# B&R Automation Studio project server
Automation Studio 4.4.6.71 SP

## Configuration minimal

### Hardware
```
X20CP1586 : X20CP1586 v1.4.2.0
  Connector IF2:
    ActivateDevice = 1
    Mode = Manual
    InternetAddress = 10.4.22.176
    SubnetMask = 255.255.255.0
  ConfigurationID = br_server_minimal
  Simulation = 1
```

## Logical view

Binary libraries used (declarations not repeated): AsBrStr, AsIecCon, AsIOTime, runtime

### Global.typ - Global data types
```iecst
TYPE
	_expData : 	STRUCT
		bActivateExperiment : BOOL;
	END_STRUCT;
	_trajData : 	STRUCT
		dStartValue : LREAL;
		lStartTime : UDINT;
		dEndValue : LREAL;
		lEndTime : UDINT;
		dOutput : LREAL;
	END_STRUCT;
	_benchData : 	STRUCT
		lTime : UDINT;
		dValue1 : LREAL;
		fValue2 : REAL;
		iValue3 : INT;
		cValue4 : BYTE;
		dValueNan : LREAL;
		dValueInf : LREAL;
	END_STRUCT;
END_TYPE
```

### Global.var - Global variables
```iecst
VAR
	expData : _expData;
	trajData : _trajData;
	benchData : _benchData;
END_VAR
```

### Package Logical/Libraries - Global libraries

### Comm.h
```c
/**
 * @file Comm.h
 */
#ifndef COMM_H
#define COMM_H

#include "Transport/Frame.h"

#define MAX_PAYLOAD (80)

/**
 * @class Comm
 * @brief defines an interface class which lets the TcpIpServer communicate with the transport protocol
 */
class Comm {
	public:
	virtual void handleFrame(Frame frame) = 0;
};

#endif
```

### TcpIpServer.h
```c
#ifndef TCPSERVER_CLASS_H
#define TCPSERVER_CLASS_H
#include <bur/plctypes.h>
#ifdef _DEFAULT_INCLUDES
#include <AsDefault.h>
#endif
#include <AsTCP.h>
#include <AsIOTime.h>
#include "../Comm.h"
#include "../Transport/Frame.h"

/** @file TcpServer.h
 *  @class TcpIpServer
 *  @brief Implementation of a simple TCP Server
 *
 *	The server is initialised and run using the BuR AsTCP library.
 */

class TcpIpServer: public Comm{
	public:
	/** server status enum */
	enum Status
	{
		ERROR = 0xFF,
		STOP = 0,
		BUSY,
		READY
	};
	private:
	const int serverPort;		///< port to be used by the server
	unsigned long serverID;		///< server ID for function blocks

	unsigned long clientIp;		///< IP address of connected client
	unsigned long clientID;		///< client ID for function blocks

	unsigned short tcp_step;		///< step variable for the server state-machine

	Status _status;
	Status _status_sub;

	struct TcpOpen TcpOpen_0;
	struct TcpServer TcpServer_0;
	struct TcpIoctl TcpIoctl_0;
	struct TcpRecv TcpRecv_0;
	struct TcpSend TcpSend_0;
	struct TcpClose TcpClose_0;

	unsigned char outBuffer[2][255 * (MAX_PAYLOAD + 1)];
	unsigned int outBufferLen[2];
	unsigned char currentOutBuf;
	unsigned char inBuffer[255 * (MAX_PAYLOAD + 1)];
	unsigned int inBufferLen;

	Status read();
	Status write();

	Comm *transp;

	public:
	TcpIpServer(int port)
		:serverPort(port),
		status(_status)
	{};

	void deinit();
	void init();
	/** cyclic read/write method */
	void sync();

	void closeSockets();
	/** readonly pointer to server status */
	const Status &status;
	/** Method to queue communication frame */
	void handleFrame(Frame frame);
	/** Method to register the transport protocol instance */
	void registerListener(Comm *transp);
};
#endif //TCPSERVER_CLASS_H
```

### Program Logical/Libraries/Transport

#### Frame.h
```c
/** @file Frame.h
 *
 */
#ifndef FRAME_H
#define FRAME_H

#include <bur/plctypes.h>
#ifdef _DEFAULT_INCLUDES
#include <AsDefault.h>
#endif
#include <stdint.h>
#include <assert.h>
#include <stdio.h>
#include <string.h>

#include "../Comm.h"

/** frame length */
#define MAX_PAYLOAD (80)

/**
 * Class, that implements a byte wise frame that is interchanged by connection. The frame has an id and a payload
 * for the specific data. The data is stored as an byte array. It implements all functions to store and unpack
 * the data to and from byte wise array. The id represents the identification of the frame.
 */
class Frame {

public:
	struct _data {
		unsigned char id;
		unsigned char payload[80];
	} data;

	Frame(unsigned char id) {
		data.id = id;
		cCursor = 0;
	}

	Frame() {
		cCursor = 0;
	}

    /** pack value into Frame
     *
     * use `pack<typename>(value)` to be explicit
     **/
	template<typename T>
	void pack(T value) {
		const unsigned int sz = sizeof(T);
		assert(cCursor + sz < MAX_PAYLOAD);
		memcpy(&data.payload[cCursor], &value, sz);
		cCursor += sz;
	}

	/** unpack into value from Frame
     *
     * use `unPack<typename>(location)` to be explicit
     */
	template<typename T>
	void unPack(T &value) {
		const unsigned int sz = sizeof(T);
		assert(cCursor + sz < MAX_PAYLOAD);
		memcpy(&value, &data.payload[cCursor], sz);
		cCursor += sz;
	}

private:
	unsigned char cCursor;

	union {
		double dVar;
		struct {
			float fVar2;
			float fVar1;
		};
		unsigned char cVar[8];
	} uPack;

};

#endif //SERVER_FRAME_H
```

#### Transport.cpp
```cpp
#define _BUR_USE_DECLARATION_IN_IEC
#ifdef _DEFAULT_INCLUDES
#include "AsDefault.h"
#endif
#include "Transport.h"

/**
 * @brief Method that defines and sends all testbench frames
 */
void Transport::sendData() {
	Frame benchFrame(10);
	benchFrame.pack(benchData.lTime);
	benchFrame.pack(benchData.dValue1);
	benchFrame.pack(benchData.fValue2);
	benchFrame.pack(benchData.iValue3);
	benchFrame.pack(benchData.cValue4);
	benchFrame.pack(benchData.dValueNan);
	benchFrame.pack(benchData.dValueInf);
	tcp->handleFrame(benchFrame);

	Frame trajFrame(11);
	trajFrame.pack(benchData.lTime);
	trajFrame.pack(trajData.dOutput);
	tcp->handleFrame(trajFrame);
}

/*
 * @brief handles all frames arriving at the testbench
 */
void Transport::handleFrame(Frame frame)
{
	switch (frame.data.id) {
		case 1:
			unpackExp(frame);
			break;
		case 12:
			unpackBenchData(frame);
			break;
		case 13:
			unpackTrajRampData(frame);
			break;
		default:;
	}
}

/**
 * @brief unpacks experiment activation status and resets experiment time
 */
void Transport::unpackExp(Frame frame) {
	frame.unPack(expData.bActivateExperiment);
	benchData.lTime = 0;
}

void Transport::unpackBenchData(Frame frame) {
	frame.unPack(benchData.dValue1);
	frame.unPack(benchData.fValue2);
	frame.unPack(benchData.iValue3);
	frame.unPack(benchData.cValue4);
}

void Transport::unpackTrajRampData(Frame frame) {
	frame.unPack(trajData.dStartValue);
	frame.unPack(trajData.lStartTime);
	frame.unPack(trajData.dEndValue);
	frame.unPack(trajData.lEndTime);
}

/**
 * @brief registers Server for handling outgoing frames
 */
void Transport::registerServer(Comm *serv)
{
	this->tcp = serv;
}
```

### Program Logical/ControlLoop (ANSIC)

#### Main.cpp - Init, cyclic, exit code
```cpp
#include <bur/plc.h>
#include <bur/plctypes.h>
#include <math.h>

#ifdef _DEFAULT_INCLUDES
	#include <AsDefault.h>
#endif

#include "../Libraries/Transport/Transport.h"

// amount of memory to be allocated for heap storage must be specified for every ANSI C++ program with the bur_heap_size variable
unsigned long bur_heap_size = 0xFFFF;
const unsigned long lDt = 1000;          ///< Sampling step [ms]

/**
 * @brief Method that calculates a trajectory value and writes the return value in _trajData->dOutput
 * @param _benchData pointer to test rig data struct
 * @param _trajData pointer to trajectory struct
 */
void fTrajectory() {
	if (benchData.lTime < trajData.lStartTime) {
		trajData.dOutput = trajData.dStartValue;
	} else {
		if (benchData.lTime < trajData.lEndTime) {
			double dM = (trajData.dEndValue - trajData.dStartValue) / (trajData.lEndTime - trajData.lStartTime);
			double dN = trajData.dEndValue - dM * trajData.lEndTime;
			trajData.dOutput = dM * benchData.lTime + dN;
		} else {
			trajData.dOutput = trajData.dEndValue;
		}
	}
}

void _INIT ProgramInit(void) {
	benchData.lTime = 0;
	benchData.dValue1 = 0;
	benchData.fValue2 = 0;
	benchData.iValue3 = 0;
	benchData.cValue4 = 0;
	benchData.dValueNan = nan("");
	benchData.dValueInf =  infinity();

	trajData.dStartValue = 0;
	trajData.lStartTime = 0;
	trajData.dEndValue = 0;
	trajData.lEndTime = 0;
	trajData.dOutput = 0;
}

void _CYCLIC ProgramCyclic(void)
{
		fTrajectory();
}

void _EXIT ProgramExit(void)
{
	// Insert code here

}
```

Listed in the project but not available here: Logical/TcpIpServer, Logical/ControlLoop/Types.typ, Logical/ControlLoop/Variables.var
